SUBAPPLICATION Counter (* Subapplication Type *)
  (* Standard: 61499-2 *)
  (* Version 1.0, 2022-12-21, Maximilian Scharf *)
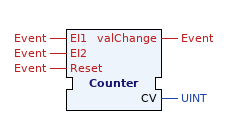
  EVENT_INPUT
    EI1;
    EI2;
    Reset;
  END_EVENT
  EVENT_OUTPUT
    valChange;
  END_EVENT
  VAR_OUTPUT
    CV : UINT;
  END_VAR
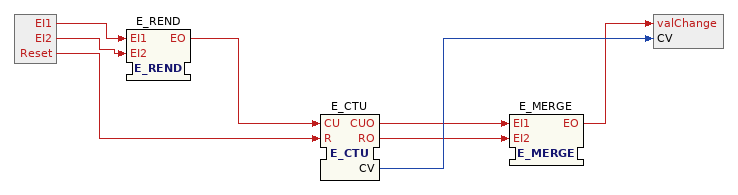
  (* Group __Group01: This subFB counts  up, starting from 0, if two different input events (EI1 and EI2) arrived and returns a valChanged event is the counter Value CV has changed. *)
  FBS
    E_MERGE : E_MERGE;
    E_CTU : E_CTU;
    E_REND : E_REND;
  END_FBS
  EVENT_CONNECTIONS
    E_CTU.CUO TO E_MERGE.EI1;
    E_CTU.RO TO E_MERGE.EI2;
    E_REND.EO TO E_CTU.CU;
    E_MERGE.EO TO valChange;
    Reset TO E_CTU.R;
    EI1 TO E_REND.EI1;
    EI2 TO E_REND.EI2;
  END_CONNECTIONS
  DATA_CONNECTIONS
    E_CTU.CV TO CV;
  END_CONNECTIONS
END_SUBAPPLICATION
